// Mitsubishi GX Works2 project: Group_10_ (2) (2)   PLC: FX3G

// global labels: Global1
VAR_GLOBAL
  X_7 AT X007 : BOOL;
  StartDay AT X007 : BOOL;
  TotalPackages AT D5555 : REAL;
END_VAR
VAR_GLOBAL CONSTANT
  ResetAnalogOutput : INT;
  ResetPackages : REAL;
END_VAR
VAR_GLOBAL
  AnalogOutput AT D8282 : INT;
  InitOatStock AT D1101 : REAL;
  OatStock AT D1111 : REAL;
  InitProteinStock AT D1103 : REAL;
  ProteinStock AT D1113 : REAL;
  InitHoneyStock AT D1105 : REAL;
  HoneyStock AT D1115 : REAL;
  WorkdayLight AT Y000 : BOOL;
  LackOfStock AT M0 : BOOL;
  EmergencySwitch AT X005 : BOOL;
  SnackTypeSample AT X003 : BOOL;
  AnalogInput1 AT D8280 : INT;
  Analog1AsFloat AT D1221 : REAL;
END_VAR
VAR_GLOBAL CONSTANT
  Divider : REAL := 400;
END_VAR
VAR_GLOBAL
  IndicatorLight AT M1 : BOOL;
END_VAR
VAR_GLOBAL CONSTANT
  ClassicSnack : REAL := 5;
END_VAR
VAR_GLOBAL
  ClassicSnackLight AT M22 : BOOL;
END_VAR
VAR_GLOBAL CONSTANT
  OatForPackage : REAL := 240;
  OatForPackageE400 : INT := 400;
  DividerE400 : INT := 400;
  ClassicSnackE5 : INT := 5;
  ProteinForPackage : REAL := 160;
  ProteinForPackageE160 : INT := 160;
  HoneyForPackageE120 : INT := 120;
END_VAR
VAR_GLOBAL
  ClassicPackageLight AT M2 : BOOL;
END_VAR
VAR_GLOBAL CONSTANT
  ProteinSnackE6 : INT := 6;
END_VAR
VAR_GLOBAL
  ProteinSnackLight AT M33 : BOOL;
END_VAR
VAR_GLOBAL CONSTANT
  OatForPackageE240 : INT := 240;
  ProteinForPackageE320 : INT := 320;
  HoneyForPackageE160 : INT := 160;
END_VAR
VAR_GLOBAL
  ProteinPackageLight AT M6 : BOOL;
  Continue AT M50 : BOOL;
  ClassicContainer AT D2000 : REAL;
END_VAR
VAR_GLOBAL CONSTANT
  ClassicContainerAddE680 : REAL := 680;
END_VAR
VAR_GLOBAL
  Container AT D2000 : REAL;
END_VAR
VAR_GLOBAL CONSTANT
  ClassicAddE680 : REAL := 680;
  ProteinAddE720 : INT := 720;
END_VAR
VAR_GLOBAL
  FinishMix AT M40 : BOOL;
  SnackTime AT TC200 : BOOL;
END_VAR
VAR_GLOBAL CONSTANT
  TotalSnackTime : INT := 500;
  TotalSnackTimeK5 : INT := 500;
END_VAR
VAR_GLOBAL
  MixingTimer AT TS200 : BOOL;
  MixingTimeLight AT Y003 : BOOL;
  DividerE4 AT E400 : REAL;
  StartMix AT M40 : BOOL;
  Baking AT X002 : BOOL;
  HelpBaking AT M60 : BOOL;
  Oven AT D2002 : REAL;
  StartBaking AT M60 : BOOL;
END_VAR
VAR_GLOBAL CONSTANT
  ClassicSnackBaking : INT := 400;
  ClassicSnackBakingK50 : INT := 40;
END_VAR
VAR_GLOBAL
  ProteinLightTime AT TC202 : BOOL;
END_VAR
VAR_GLOBAL CONSTANT
  ProteinSnackBakingK30 : INT := 50;
  ProteinSnackBakingK50 : INT := 500;
  ClassicSnackBakingK40 : INT := 400;
END_VAR
VAR_GLOBAL
  ProteinLightTime1 AT TS202 : BOOL;
  HelpLight AT M5 : BOOL;
  FirstLightTime AT TC203 : BOOL;
  FirstLight AT Y001 : BOOL;
END_VAR
VAR_GLOBAL CONSTANT
  FlickerTime : INT := 50;
  FlickerTimeK05 : INT := 50;
END_VAR
VAR_GLOBAL
  FirstLightTimer AT TS203 : BOOL;
  SecondLightTimer AT TS204 : BOOL;
  SecondLight AT Y002 : BOOL;
  SecondLightTime AT TC204 : BOOL;
  StartPacking AT X006 : BOOL;
  OneSnackPacking AT X000 : BOOL;
  SnackCounter AT CC0 : BOOL;
END_VAR
VAR_GLOBAL CONSTANT
  FirstSnackK1 : INT := 1;
  FullPackageK8 : INT := 8;
END_VAR
VAR_GLOBAL
  PackageCounter AT CC1 : BOOL;
  StartSnackPacking AT X000 : BOOL;
  FinishSnackPacking AT CS0 : BOOL;
  FinishPackagePacking AT CS1 : BOOL;
  PackingLight AT Y004 : BOOL;
END_VAR
VAR_GLOBAL CONSTANT
  NewPackageE1 : INT := 1;
END_VAR
VAR_GLOBAL
  IterationLight AT M100 : BOOL;
END_VAR
VAR_GLOBAL CONSTANT
  MultipleE40 : INT := 40;
  Reset : REAL;
END_VAR
VAR_GLOBAL
  SaveAnalogInput1 AT D8201 : INT;
END_VAR
VAR_GLOBAL CONSTANT
  HoneyForPackage : REAL := 120;
  ProteinSnack : REAL := 6;
  OatForClassicPackage : REAL := 400;
  ProteinForClassicPackage : REAL := 160;
  HoneyForClassicPackage : REAL := 120;
  OatForProteinPackage : REAL := 240;
  ProteinForProteinPackage : REAL := 320;
  HoneyForProteinPackage : REAL := 160;
  ClassicAdd : REAL := 680;
  ProteinAdd : REAL := 720;
  ProteinSnackBaking : INT := 500;
  FirstSnack : INT := 1;
  FullPackage : INT := 8;
  NewPackage : REAL := 1;
  Multiple : REAL := 40;
END_VAR
VAR_GLOBAL
  ClassicLightTime AT TS201 : BOOL;
END_VAR

// task Task_01 (event TRUE, interval 0, priority 31): POU_01

PROGRAM POU_01
(* structured ladder/FBD written out as ST: instructions are called as NAME(EN, inputs, outputs); _pN, _eN, _tN stand for wires *)
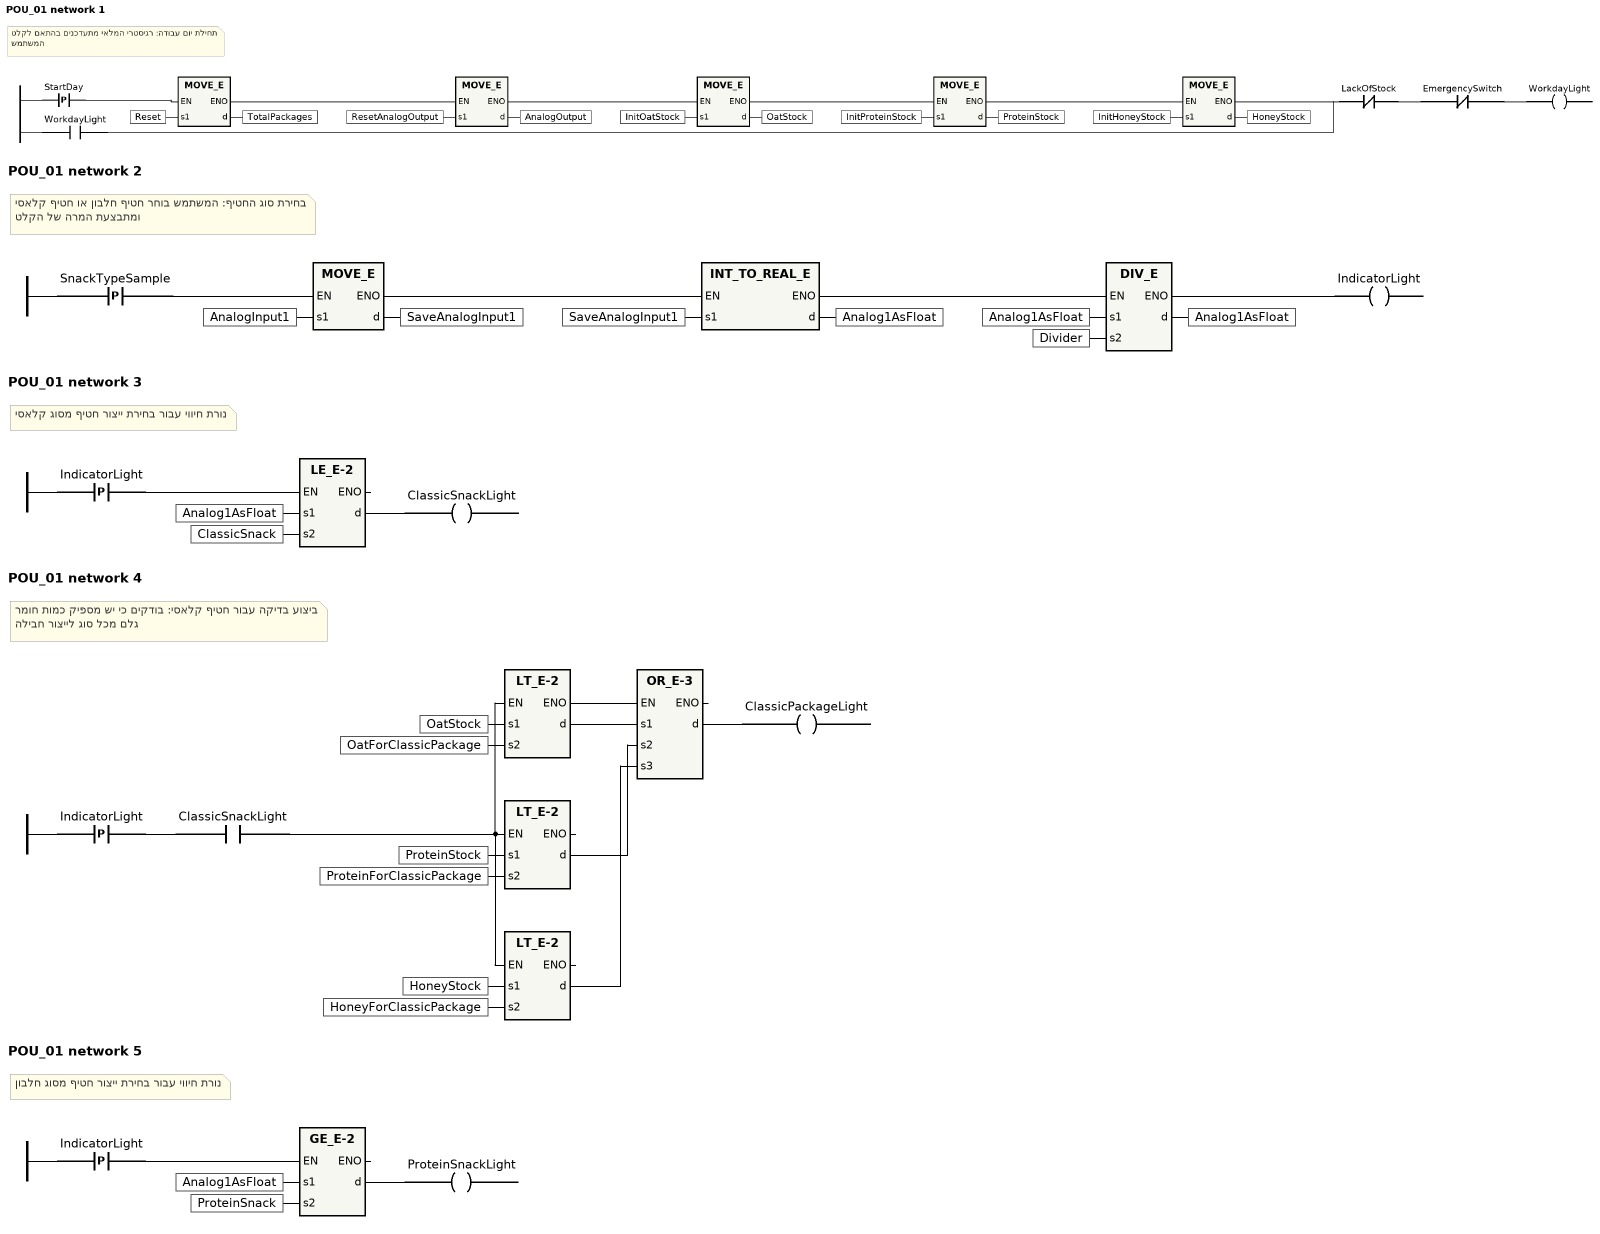
(* network 1 *)
(* תחילת יום עבודה: רגיסטרי המלאי מתעדכנים בהתאם לקלט המשתמש *)
_e1 := MOVE_E(LDP(TRUE, StartDay), Reset, TotalPackages);
_e2 := MOVE_E(_e1, ResetAnalogOutput, AnalogOutput);
_e3 := MOVE_E(_e2, InitOatStock, OatStock);
_e4 := MOVE_E(_e3, InitProteinStock, ProteinStock);
_e5 := MOVE_E(_e4, InitHoneyStock, HoneyStock);
WorkdayLight := ((_e5 OR WorkdayLight) AND NOT LackOfStock) AND NOT EmergencySwitch;
(* network 2 *)
(* בחירת סוג החטיף: המשתמש בוחר חטיף חלבון או חטיף קלאסי ומתבצעת המרה של הקלט *)
_e1 := MOVE_E(LDP(TRUE, SnackTypeSample), AnalogInput1, SaveAnalogInput1);
_e2 := INT_TO_REAL_E(_e1, SaveAnalogInput1, Analog1AsFloat);
_e3 := DIV_E(_e2, Analog1AsFloat, Divider, Analog1AsFloat);
IndicatorLight := _e3;
(* network 3 *)
(* נורת חיווי עבור בחירת ייצור חטיף מסוג קלאסי *)
LE_E(LDP(TRUE, IndicatorLight), Analog1AsFloat, ClassicSnack, _t1);
ClassicSnackLight := _t1;
(* network 4 *)
(* ביצוע בדיקה עבור חטיף קלאסי: בודקים כי יש מספיק כמות חומר גלם מכל סוג לייצור חבילה *)
_p1 := LDP(TRUE, IndicatorLight) AND ClassicSnackLight;
_e3 := LT_E(_p1, OatStock, OatForClassicPackage, _t2);
LT_E(_p1, ProteinStock, ProteinForClassicPackage, _t4);
LT_E(_p1, HoneyStock, HoneyForClassicPackage, _t5);
OR_E(_e3, _t2, _t4, _t5, _t6);
ClassicPackageLight := _t6;
(* network 5 *)
(* נורת חיווי עבור בחירת ייצור חטיף מסוג חלבון *)
GE_E(LDP(TRUE, IndicatorLight), Analog1AsFloat, ProteinSnack, _t1);
ProteinSnackLight := _t1;
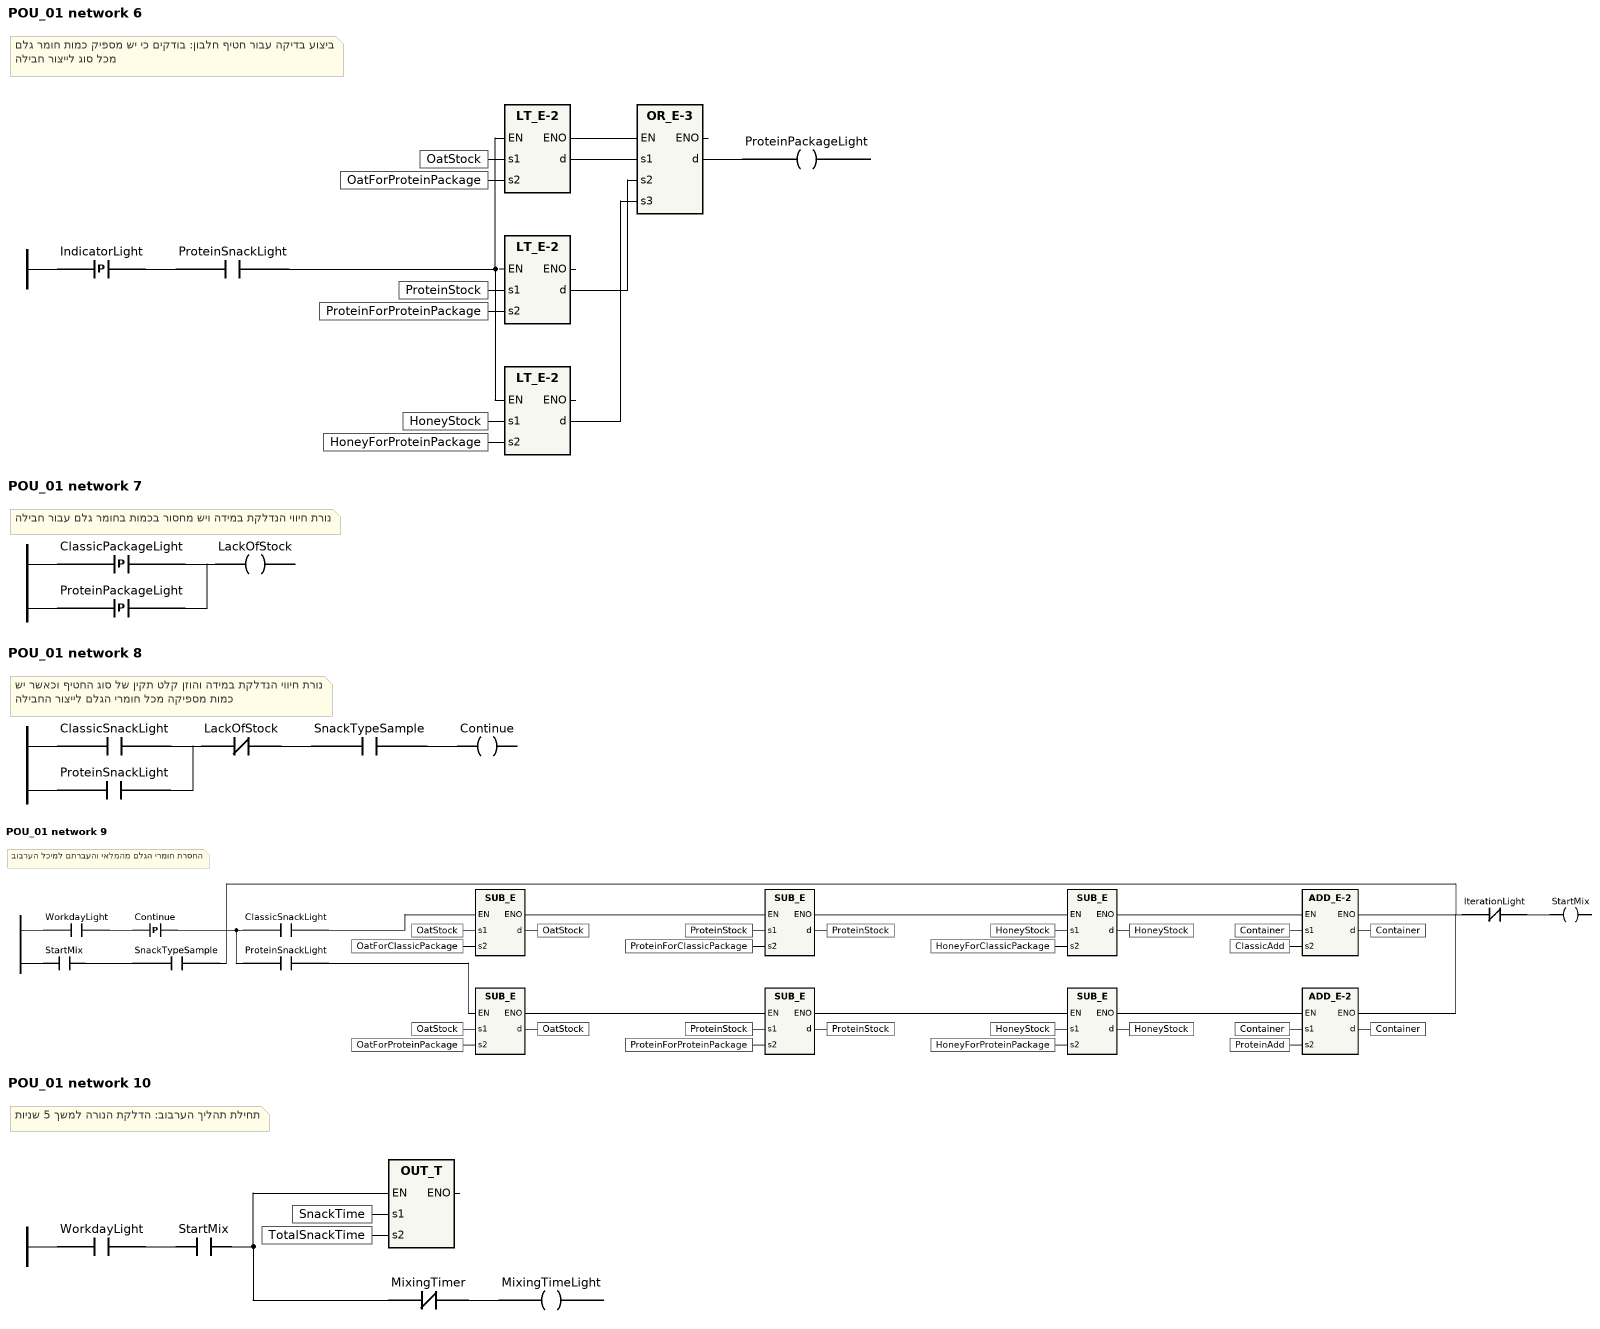
(* network 6 *)
(* ביצוע בדיקה עבור חטיף חלבון: בודקים כי יש מספיק כמות חומר גלם מכל סוג לייצור חבילה *)
_p1 := LDP(TRUE, IndicatorLight) AND ProteinSnackLight;
_e3 := LT_E(_p1, OatStock, OatForProteinPackage, _t2);
LT_E(_open, ProteinStock, ProteinForProteinPackage, _t4);
LT_E(_p1, HoneyStock, HoneyForProteinPackage, _t5);
OR_E(_e3, _t2, _t4, _t5, _t6);
ProteinPackageLight := _t6;
(* network 7 *)
(* נורת חיווי הנדלקת במידה ויש מחסור בכמות בחומר גלם עבור חבילה *)
LackOfStock := LDP(TRUE, ClassicPackageLight) OR LDP(TRUE, ProteinPackageLight);
(* network 8 *)
(* נורת חיווי הנדלקת במידה והוזן קלט תקין של סוג החטיף וכאשר יש כמות מספיקה מכל חומרי הגלם לייצור החבילה *)
Continue := ((ClassicSnackLight OR ProteinSnackLight) AND NOT LackOfStock) AND SnackTypeSample;
(* network 9 *)
(* החסרת חומרי הגלם מהמלאי והעברתם למיכל הערבוב *)
_p1 := WorkdayLight AND LDP(TRUE, Continue);
_e2 := SUB_E(_p1 AND ClassicSnackLight, OatStock, OatForClassicPackage, OatStock);
_e3 := SUB_E(_e2, ProteinStock, ProteinForClassicPackage, ProteinStock);
_e4 := SUB_E(_e3, HoneyStock, HoneyForClassicPackage, HoneyStock);
_e5 := ADD_E(_e4, Container, ClassicAdd, Container);
_e6 := SUB_E(_p1 AND ProteinSnackLight, OatStock, OatForProteinPackage, OatStock);
_e7 := SUB_E(_e6, ProteinStock, ProteinForProteinPackage, ProteinStock);
_e8 := SUB_E(_e7, HoneyStock, HoneyForProteinPackage, HoneyStock);
_e9 := ADD_E(_e8, Container, ProteinAdd, Container);
StartMix := (_e5 OR _e9 OR (StartMix AND SnackTypeSample)) AND NOT IterationLight;
(* network 10 *)
(* תחילת תהליך הערבוב: הדלקת הנורה למשך 5 שניות *)
_p1 := WorkdayLight AND StartMix;
OUT_T(_p1, SnackTime, TotalSnackTime);
MixingTimeLight := _p1 AND NOT MixingTimer;
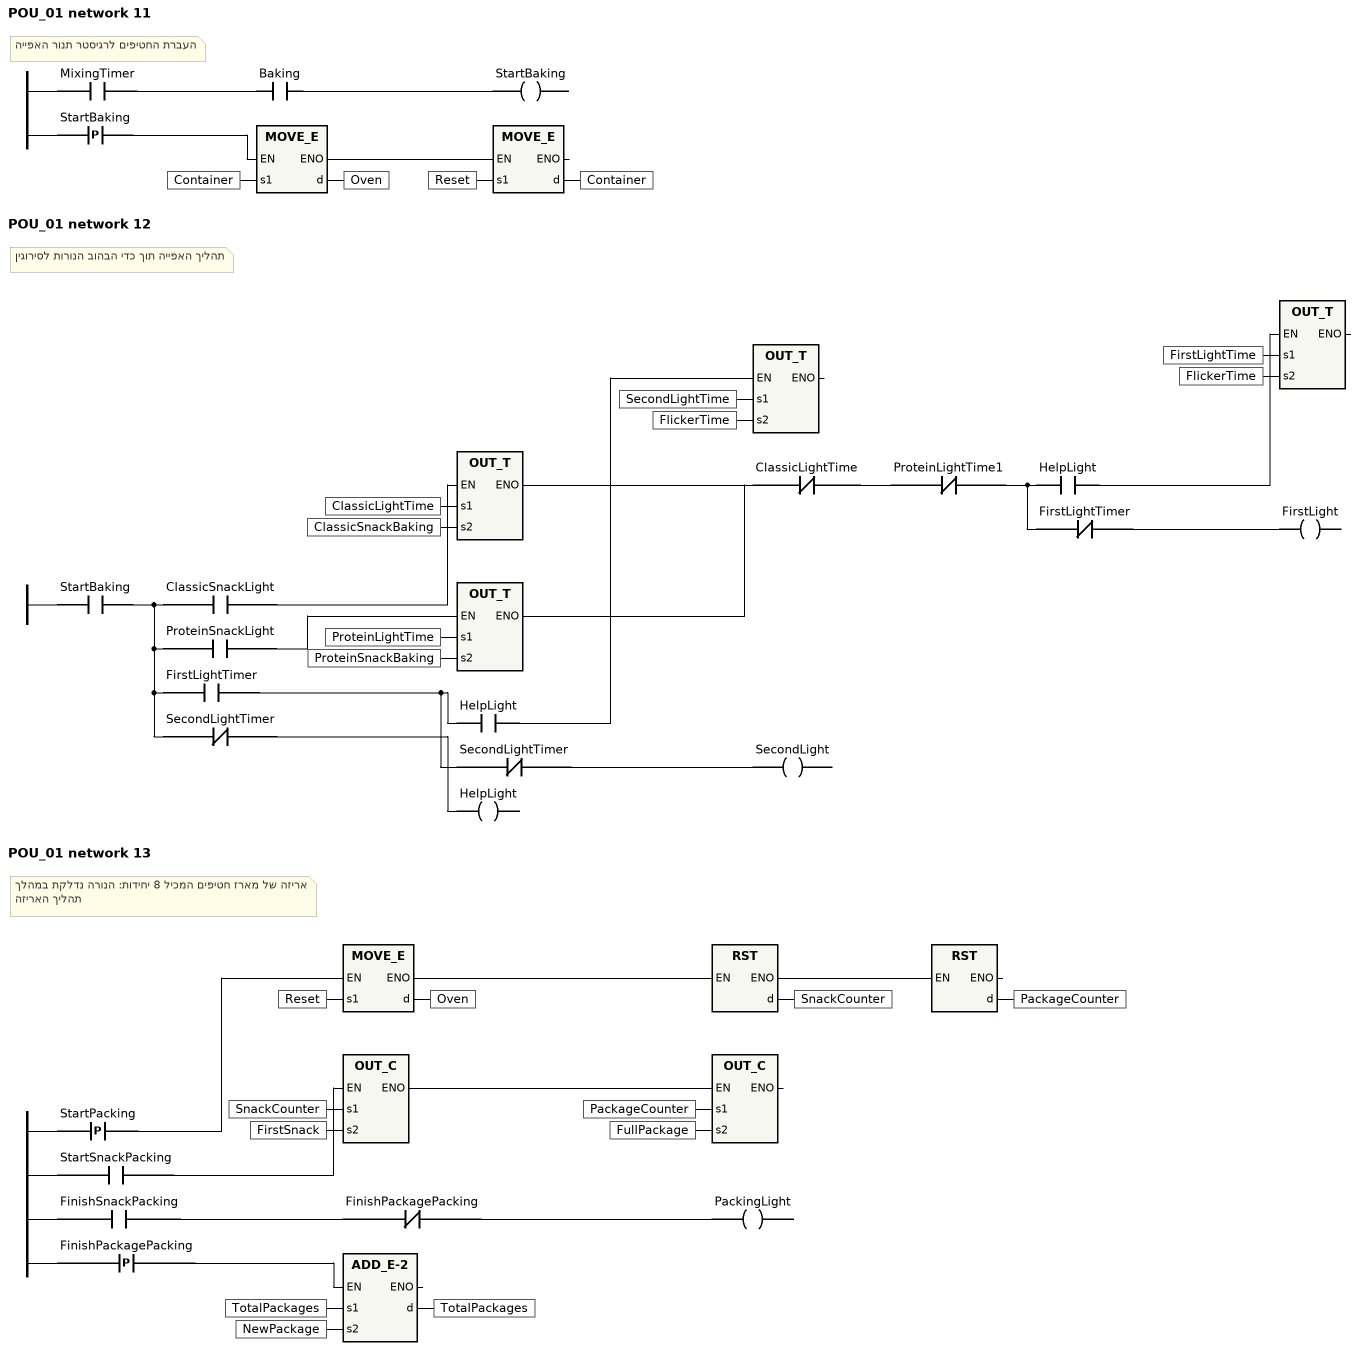
(* network 11 *)
(* העברת החטיפים לרגיסטר תנור האפייה *)
StartBaking := MixingTimer AND Baking;
_e1 := MOVE_E(LDP(TRUE, StartBaking), Container, Oven);
MOVE_E(_e1, Reset, Container);
(* network 12 *)
(* תהליך האפייה תוך כדי הבהוב הנורות לסירוגין *)
_e1 := OUT_T(StartBaking AND ClassicSnackLight, ClassicLightTime, ClassicSnackBaking);
_e2 := OUT_T(StartBaking AND ProteinSnackLight, ProteinLightTime, ProteinSnackBaking);
_p3 := ((_e1 OR _e2) AND NOT ClassicLightTime) AND NOT ProteinLightTime1;
OUT_T(_p3 AND HelpLight, FirstLightTime, FlickerTime);
FirstLight := _p3 AND NOT FirstLightTimer;
_p4 := StartBaking AND FirstLightTimer;
OUT_T(_p4 AND HelpLight, SecondLightTime, FlickerTime);
SecondLight := _p4 AND NOT SecondLightTimer;
HelpLight := StartBaking AND NOT SecondLightTimer;
(* network 13 *)
(* אריזה של מארז חטיפים המכיל 8 יחידות: הנורה נדלקת במהלך תהליך האריזה *)
_e1 := MOVE_E(LDP(TRUE, StartPacking), Reset, Oven);
_e2 := RST(_e1, SnackCounter);
RST(_e2, PackageCounter);
_e3 := OUT_C(StartSnackPacking, SnackCounter, FirstSnack);
OUT_C(_e3, PackageCounter, FullPackage);
PackingLight := FinishSnackPacking AND NOT FinishPackagePacking;
ADD_E(LDP(TRUE, FinishPackagePacking), TotalPackages, NewPackage, TotalPackages);
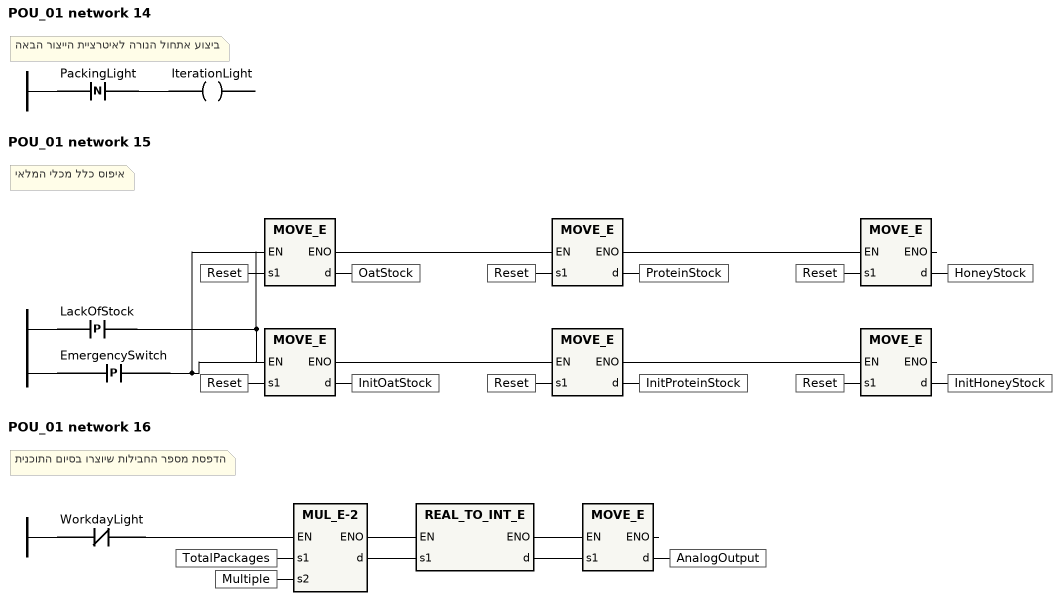
(* network 14 *)
(* ביצוע אתחול הנורה לאיטרציית הייצור הבאה *)
IterationLight := LDF(TRUE, PackingLight);
(* network 15 *)
(* איפוס כלל מכלי המלאי *)
_p1 := LDP(TRUE, LackOfStock) OR LDP(TRUE, EmergencySwitch);
_e2 := MOVE_E(_p1, Reset, OatStock);
_e3 := MOVE_E(_e2, Reset, ProteinStock);
MOVE_E(_e3, Reset, HoneyStock);
_e4 := MOVE_E(_p1, Reset, InitOatStock);
_e5 := MOVE_E(_e4, Reset, InitProteinStock);
MOVE_E(_e5, Reset, InitHoneyStock);
(* network 16 *)
(* הדפסת מספר החבילות שיוצרו בסיום התוכנית *)
_e2 := MUL_E(NOT WorkdayLight, TotalPackages, Multiple, _t1);
_e4 := REAL_TO_INT_E(_e2, _t1, _t3);
MOVE_E(_e4, _t3, AnalogOutput);
END_PROGRAM
